Omron CX-Programmer project NewProject (CX-Programmer 9.81)

# PLC NewPLC1: CJ1M CPU11
I/O table (CPU CJ1M-CPU11): rack 0 slot 0 CJ1W-ID211; rack 0 slot 1 CJ1W-OD211

## Program NewProgram1 (cyclic task 0)
Local symbols
KM1 1.00 BOOL  ; Andar para a direita
KM2 1.01 BOOL  ; Anda para a esquerda
Led_Start 1.03 BOOL  ; Led start
S_P 0.03 BOOL  ; Sensor de peso
S_a 0.01 BOOL  ; fim de curso A
S_b 0.02 BOOL  ; Fim de curso B
V1 1.02 BOOL  ; Valvula
b_s 0.00 BOOL  ; Botão Start
etapa_0 2.00 BOOL  ; Ligar o Led
etapa_1 2.01 BOOL  ; Andar para a Direita
etapa_2 2.02 BOOL  ; Parar de andar para a direita e abrir a valvula
etapa_3 2.03 BOOL  ; Fechar a valvula e andar para a esquerda
etapa_4 2.04 BOOL  ; para de andar para a esquerda

### Section MAIN

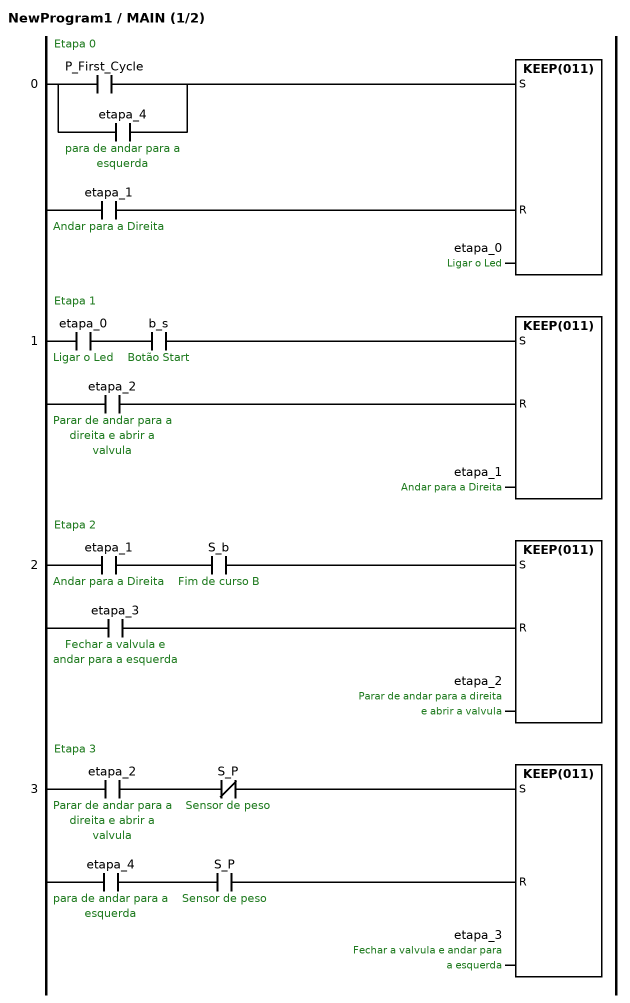
; rung 0: Etapa 0
LD P_First_Cycle
OR etapa_4  ; para de andar para a esquerda
LD etapa_1  ; Andar para a Direita
KEEP(011) etapa_0  ; Ligar o Led
; rung 1: Etapa 1
LD etapa_0  ; Ligar o Led
AND b_s  ; Botão Start
LD etapa_2  ; Parar de andar para a direita e abrir a valvula
KEEP(011) etapa_1  ; Andar para a Direita
; rung 2: Etapa 2
LD etapa_1  ; Andar para a Direita
AND S_b  ; Fim de curso B
LD etapa_3  ; Fechar a valvula e andar para a esquerda
KEEP(011) etapa_2  ; Parar de andar para a direita e abrir a valvula
; rung 3: Etapa 3
LD etapa_2  ; Parar de andar para a direita e abrir a valvula
ANDNOT S_P  ; Sensor de peso
LD etapa_4  ; para de andar para a esquerda
AND S_P  ; Sensor de peso
KEEP(011) etapa_3  ; Fechar a valvula e andar para a esquerda

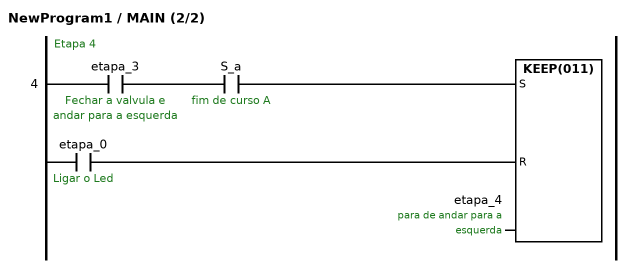
; rung 4: Etapa 4
LD etapa_3  ; Fechar a valvula e andar para a esquerda
AND S_a  ; fim de curso A
LD etapa_0  ; Ligar o Led
KEEP(011) etapa_4  ; para de andar para a esquerda

### Section OUTPUTS

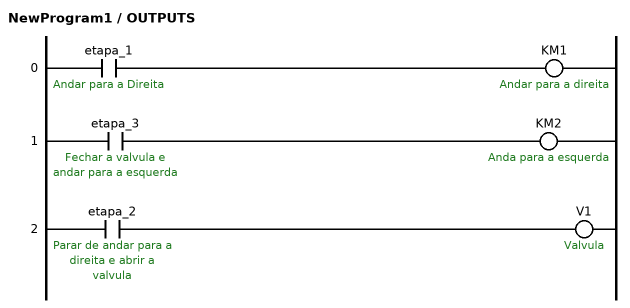
; rung 0
LD etapa_1  ; Andar para a Direita
OUT KM1  ; Andar para a direita
; rung 1
LD etapa_3  ; Fechar a valvula e andar para a esquerda
OUT KM2  ; Anda para a esquerda
; rung 2
LD etapa_2  ; Parar de andar para a direita e abrir a valvula
OUT V1  ; Valvula

### Section END
; rung 0
END(001)